Staubli VAL3: decodeMsgHeader.pgx

public program decodeMsgHeader(RosSimpleMsg& x_msg, num& x_nMsgRecvState)
  local num l_nRetVal
begin
  // Copyright (c) 2016, Ocado Technology - Robotics Research Team
  // Copyright (c) 2021, Institute for Factory Automation and Production Systems (FAPS)
  //
  // Licensed under the Apache License, Version 2.0 (the "License");
  // you may not use this file except in compliance with the License.
  // You may obtain a copy of the License at
  //
  //     http://www.apache.org/licenses/LICENSE-2.0
  //
  // Unless required by applicable law or agreed to in writing, software
  // distributed under the License is distributed on an "AS IS" BASIS,
  // WITHOUT WARRANTIES OR CONDITIONS OF ANY KIND, either express or implied.
  // See the License for the specific language governing permissions and
  // limitations under the License.



  // decode message into generic message first
  l_nRetVal=fromBinary(x_msg.prefix.nData,4,"-4l",x_msg.prefix.nLength)
  if (l_nRetVal!=1)
    // error decoding prefix, reset state machine
    x_nMsgRecvState = MsgRecvState.RECEIVE_HEADER
    return
  endIf
  l_nRetVal=fromBinary(x_msg.header.nData,4,"-4l",x_msg.header.nMsgType)
  if (l_nRetVal!=1)
    // error decoding header (msg type), reset state machine
    x_nMsgRecvState = MsgRecvState.RECEIVE_HEADER
    return
  endIf
  l_nRetVal=fromBinary(x_msg.header.nData[4],4,"-4l",x_msg.header.nCommType)
  if (l_nRetVal!=1)
    // error decoding header (comm type), reset state machine
    x_nMsgRecvState = MsgRecvState.RECEIVE_HEADER
    return
  endIf
  l_nRetVal=fromBinary(x_msg.header.nData[8],4,"-4l",x_msg.header.nReplyCode)
  if (l_nRetVal!=1)
    // error decoding header (reply code), reset state machine
    x_nMsgRecvState = MsgRecvState.RECEIVE_HEADER
    return
  endIf

  // no errors detected whilst decoding prefix and header
  // move on to state 2: receive msg body
  x_nMsgRecvState = MsgRecvState.RECEIVE_BODY

  // debug
  if (bDebugMode and nDebugLevel<=1)
    //call printDebug("decodeMsgHeader: successful",true)
    //call printDebug("Prefix    :"+toString("",x_msg.prefix.nLength),false)
    //call printDebug("MsgType   :"+toString("",x_msg.header.nMsgType),false)
    //call printDebug("CommType  :"+toString("",x_msg.header.nCommType),false)
    //call printDebug("ReplyType :"+toString("",x_msg.header.nReplyCode),false)
  endIf
end
